INTERFACE I_Testbase extends __SYSTEM.IQueryInterface

PROPERTY PUBLIC P_Name : STRING(255)
GET
END_GET
SET
END_SET
END_PROPERTY

END_INTERFACE

(* stored: Version 1.1.0.1
   Itf I_Testbase: Id {ada3f4ee-e52c-4b2e-ad47-2676c314edf3}
   Property P_Name: Id {28191297-7659-4cca-b8fa-d5c22b1395c0}
   Get Get: Id {bd54a2cd-0fa9-484e-9c8d-9f58bb8389e9}
   Set Set: Id {fb742643-9971-4b3c-ac1b-cd31488bfda0} *)
